// SIMATIC S7-200 project (STEP 7-Micro/WIN), CPU 226 CN REL 02.01

ORGANIZATION_BLOCK 主程序:OB1
TITLE=程序注释
BEGIN
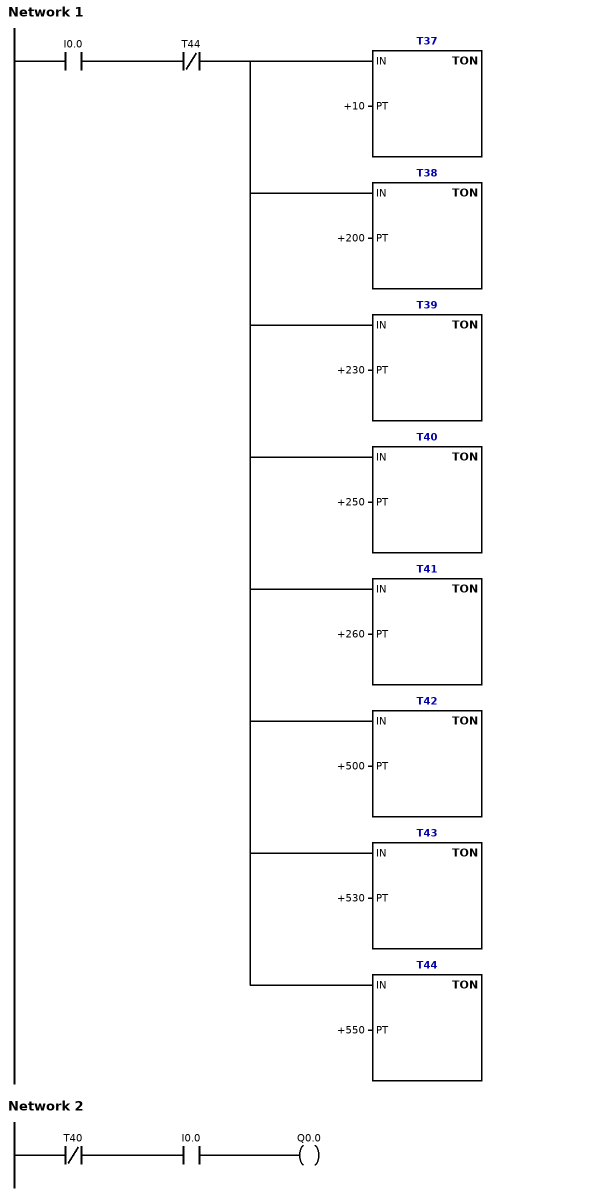
Network 1
LD     I0.0
AN     T44
TON    T37, +10
TON    T38, +200
TON    T39, +230
TON    T40, +250
TON    T41, +260
TON    T42, +500
TON    T43, +530
TON    T44, +550
Network 2
LDN    T40
A      I0.0
=      Q0.0
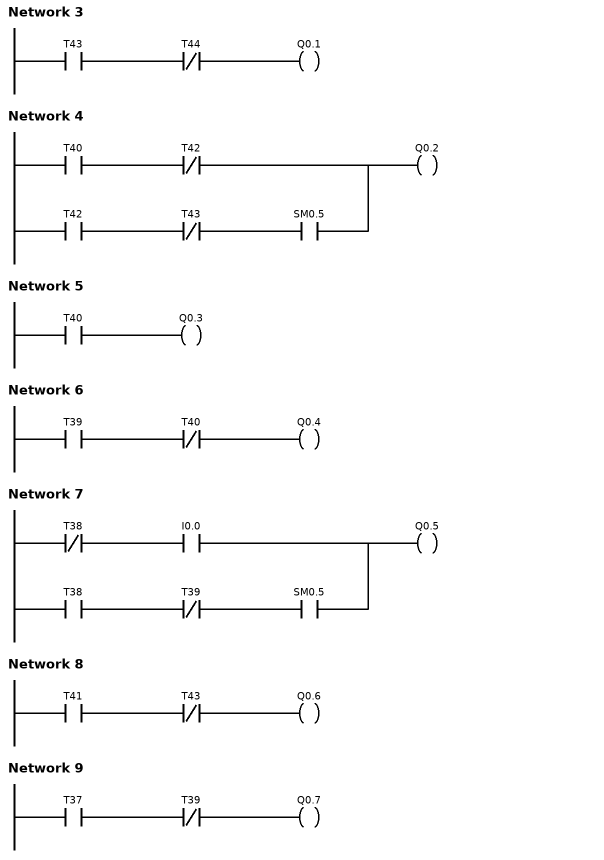
Network 3
LD     T43
AN     T44
=      Q0.1
Network 4
LD     T40
AN     T42
LD     T42
AN     T43
A      SM0.5
OLD
=      Q0.2
Network 5
LD     T40
=      Q0.3
Network 6
LD     T39
AN     T40
=      Q0.4
Network 7
LDN    T38
A      I0.0
LD     T38
AN     T39
A      SM0.5
OLD
=      Q0.5
Network 8
LD     T41
AN     T43
=      Q0.6
Network 9
LD     T37
AN     T39
=      Q0.7
END_ORGANIZATION_BLOCK
